(* IEC 61131-3 sources: xPLCCore/codesys_code/Application/COMM_FBs, 10 files *)

(* ---- E_MpParserInternalState.st ---- *)
(* Internal states for byte-by-byte parsing *)
TYPE E_MpParserInternalState :
(
	STATE_IDLE, 			// Waiting for first byte of a new item
	STATE_READING_LENGTH, 	// Reading length/count bytes
	STATE_READING_DATA 		// Reading actual payload data (skipping it)
);
END_TYPE

(* ---- E_MpType.st ---- *)
TYPE E_MpType :
(
	MP_UNKNOWN,
	MP_NIL,
	MP_BOOL,
	MP_DINT,
	MP_REAL,
	MP_STRING,
	MP_BINARY,
	MP_ARRAY,
	MP_MAP
);
END_TYPE

(* ---- E_MsgPakLevelParser_ERROR.st ---- *)
(* ============================================================================
   Error Enumeration for FB_MsgPakLevelParser
   ============================================================================ *)

TYPE E_MsgPakLevelParser_ERROR :
(
    NONE := 0,              (* No error *)
    UNEXPECTED_BYTE := 1,   (* Invalid MessagePack type byte *)
    STACK_OVERFLOW := 2,    (* Too many nested containers *)
    INVALID_STATE := 3      (* Internal parser state error *)
);
END_TYPE

(* ---- E_MsgPakLevelParser_STATE.st ---- *)
(* ============================================================================
   State Enumeration for FB_MsgPakLevelParser State Machine
   ============================================================================ *)

TYPE E_MsgPakLevelParser_STATE :
(
    EXPECT_HEADER := 0,     (* Waiting for a new MessagePack type byte *)
    EXPECT_LENGTH := 1,     (* Accumulating length bytes for variable-length types *)
    EXPECT_EXT_TYPE := 2,   (* Waiting for extension type byte *)
    EXPECT_DATA := 3        (* Consuming data bytes (strings, binaries, etc.) *)
);
END_TYPE

(* ---- T_NestingContext.st ---- *)
TYPE T_NestingContext :
STRUCT
	bIsMap 		: BOOL; // TRUE if this level is a map, FALSE if it's an array
	uiItemsLeft : UINT; // Number of items remaining to be skipped at this level
END_STRUCT
END_TYPE

(* ---- F_BYTE_TO_HEX_STRING.st ---- *)
(*
FUNCTION F_BYTE_TO_HEX_STRING
Description: Converts a single BYTE value to its two-character hexadecimal STRING representation.
             E.g., 16#0A -> '0A', 16#FF -> 'FF'
*)
FUNCTION F_BYTE_TO_HEX_STRING : STRING(2)
VAR_INPUT
	byValue : BYTE; // The byte value to convert
END_VAR
VAR CONSTANT
    HEX_CHARS : ARRAY[0..15] OF STRING(1) := ['0', '1', '2', '3', '4', '5', '6', '7', '8', '9', 'A', 'B', 'C', 'D', 'E', 'F'];
END_VAR
VAR
	byHighNibble: BYTE;
	byLowNibble : BYTE;
END_VAR
(* =========== IMPLEMENTATION =========== *)

	// Get the high nibble (upper 4 bits)
	byHighNibble := SHR(byValue, 4) AND 16#0F;
	// Get the low nibble (lower 4 bits)
	byLowNibble := byValue AND 16#0F;

	// Use array lookup for hexadecimal characters and concatenate them
	F_BYTE_TO_HEX_STRING := CONCAT(HEX_CHARS[BYTE_TO_INT(byHighNibble)], HEX_CHARS[BYTE_TO_INT(byLowNibble)]);

(* ---- F_E_MpType_TO_STRING.st ---- *)
(*
FUNCTION F_E_MpType_TO_STRING
Description: Converts an E_MpType enumeration value to its string representation.
*)
FUNCTION F_E_MpType_TO_STRING : STRING
VAR_INPUT
	eType : E_MpType; // The enumeration value to convert
END_VAR
(* =========== IMPLEMENTATION =========== *)

	CASE eType OF
		E_MpType.MP_UNKNOWN:
			F_E_MpType_TO_STRING := 'UNKNOWN';
		E_MpType.MP_NIL:
			F_E_MpType_TO_STRING := 'NIL';
		E_MpType.MP_BOOL:
			F_E_MpType_TO_STRING := 'BOOL';
		E_MpType.MP_DINT:
			F_E_MpType_TO_STRING := 'DINT';
		E_MpType.MP_REAL:
			F_E_MpType_TO_STRING := 'REAL';
		E_MpType.MP_STRING:
			F_E_MpType_TO_STRING := 'STRING';
		E_MpType.MP_BINARY:
			F_E_MpType_TO_STRING := 'BINARY';
		E_MpType.MP_ARRAY:
			F_E_MpType_TO_STRING := 'ARRAY';
		E_MpType.MP_MAP:
			F_E_MpType_TO_STRING := 'MAP';
		ELSE
			F_E_MpType_TO_STRING := 'ERROR_INVALID_TYPE';
	END_CASE;

(* ---- Swap16To.st ---- *)
FUNCTION Swap16To : BOOL // Or VOID if your CoDeSys version supports it for functions
VAR_INPUT
	srcData : POINTER TO BYTE;
	dstData : POINTER TO BYTE;
END_VAR
VAR
END_VAR
(* =========== IMPLEMENTATION =========== *)

	// Check for a valid pointer (optional but good practice)
	IF dstData = 0 OR srcData=0 THEN
		Swap16To := FALSE;
		RETURN;
	END_IF;

	dstData[0]:=srcData[1];
	dstData[1]:=srcData[0];

	Swap16To := TRUE; // Indicate successful swap

(* ---- Swap32To.st ---- *)
FUNCTION Swap32To : BOOL // Or VOID if your CoDeSys version supports it for functions
VAR_INPUT
	srcData : POINTER TO BYTE;
	dstData : POINTER TO BYTE;
END_VAR
VAR
END_VAR
(* =========== IMPLEMENTATION =========== *)

	// Check for a valid pointer (optional but good practice)
	IF dstData = 0 OR srcData=0 THEN
		Swap32To := FALSE;
		RETURN;
	END_IF;

	dstData[0]:=srcData[3];
	dstData[3]:=srcData[0];

	dstData[1]:=srcData[2];
	dstData[2]:=srcData[1];

	Swap32To := TRUE; // Indicate successful swap

(* ---- Swap64To.st ---- *)
FUNCTION Swap64To : BOOL
VAR_INPUT
	srcData : POINTER TO BYTE; // Pointer to the source 8-byte data
	dstData : POINTER TO BYTE; // Pointer to the destination 8-byte data
END_VAR
VAR
END_VAR
(* =========== IMPLEMENTATION =========== *)

	IF dstData = 0 OR srcData = 0 THEN
		Swap64To := FALSE;
		RETURN;
	END_IF;

	// srcData (big-endian): [0][1][2][3][4][5][6][7]
	// dstData (little-endian): [7][6][5][4][3][2][1][0]
	dstData[0] := srcData[7];
	dstData[1] := srcData[6];
	dstData[2] := srcData[5];
	dstData[3] := srcData[4];
	dstData[4] := srcData[3];
	dstData[5] := srcData[2];
	dstData[6] := srcData[1];
	dstData[7] := srcData[0];

	Swap64To := TRUE;
